INTERFACE I_NodeFactoryVisitor

METHOD VisitNodeFactory
VAR_INPUT
	VisitingPrototypes : I_NodeFactory;
END_VAR
END_METHOD

END_INTERFACE

(* stored: Version 1.1.0.1, ProductVersion 3.1.4024.12
   Itf I_NodeFactoryVisitor: Id {ff1ddfce-f575-418a-a47c-82173358b9f2}
   Method VisitNodeFactory: Id {da9fe5cc-6f41-4808-861d-192c4ebbec8c} *)
